// TIA Portal V20 export
// export: Created 2025-12-01T14:57:45.1353777Z, ExportSetting None, DisplayName Totally Integrated Automation Portal, DisplayVersion V20 Update 3, DisplayName TIA Portal Openness, DisplayVersion V20 Update 3, DisplayName TIA Portal Version Control Interface, DisplayVersion V20 Update 3, DisplayName STEP 7 Professional, DisplayVersion V20 Update 3, DisplayName STEP 7 Safety, DisplayVersion V20 Update 2, DisplayName WinCC Basic/Comfort/Advanced, DisplayVersion V20 Update 3, DisplayName WinCC Professional, DisplayVersion V20 Update 3, DisplayName WinCC Unified, DisplayVersion V20 Update 3
FUNCTION "FC783_Evento_BOET" : Void   // FC783, LAD
{ S7_Optimized_Access := 'FALSE' }
// stored: AutoNumber false, SetENOAutomatically false
   VAR_INPUT
      mensaje : Int;   // indice del array que estamos extrayendo
   END_VAR
   VAR_TEMP
      cero : Byte;
      retval : Int;
      pos_SSCC : UInt;
      Etiqueta_a_eliminar : ULInt;
      posicion_a_eliminar : UInt;
      cola : UInt;
      dato_actual_cola : UInt;
      pos_DB : UInt;
      registro_anterior : UInt;
      registro_siguiente : UInt;
      registro_etiqueta_limpio : "ROUT_Reg_Etiqueta";
   END_VAR
BEGIN

REGION Network 1 (SCL): INICIALIZACIONES
   REGION inicializacion

       // inicializamos las variables
       // 

       #retval := FILL(BVAL := #cero, BLK => #registro_etiqueta_limpio); // el registro de la etiqueta temporal



   END_REGION
END_REGION

REGION Network 2 (SCL): RECOJO Y CONVIERTO EL VALOR DE LA EITQUETA
   // buscamos donde empieza el SSCC en el mensaje y lo convertimos
   // 
   #pos_SSCC := FIND(IN1 := "DB199_eventos_convertidos".evento[#mensaje], IN2 := '[SSCC]');

   STRG_VAL(IN := "DB199_eventos_convertidos".evento[#mensaje],
            FORMAT := 0,
            P := (#pos_SSCC + 6), // +6 por lo que ocupa el atributo ['SSCC]'
            OUT => #Etiqueta_a_eliminar
   );

   // buscamos la etiqueta en la BBDD

   "FC715_Router_BuscarEtiqueta_Lint"(Etiqueta :=#Etiqueta_a_eliminar ,
                                      Posicion_BBDD => #posicion_a_eliminar);


   // si la posición a eliminar es 0, es que no existe ya en la BBDD y salimos de la función
   // 
   IF #posicion_a_eliminar = 0 THEN
       RETURN;
   END_IF;

     // si la hemos encontrado, además de eliminar la etiqueta, tenemos que mantener la coherencia
     // en el sistema de colas
     // para eso tenemos que mirar la posicón anterior y siguiente
     // 
     //
     //CALCULAMOS LA COLA A LA QUE PERTENECE LA ETIQUETA 
   #cola :=#Etiqueta_a_eliminar MOD "ROUT_N_Colas";


   REGION elegir_db_busqueda
       CASE #posicion_a_eliminar OF
           1..1000:
               #pos_DB := #posicion_a_eliminar;
               #registro_anterior:="DB201_RegEtiquetas_0001_1000".Reg_Etiqueta[#pos_DB].Anterior;
               #registro_siguiente:="DB201_RegEtiquetas_0001_1000".Reg_Etiqueta[#pos_DB].Posterior;
               // ahora que ya he sacado los datos necesarios limpio el registro
               "DB201_RegEtiquetas_0001_1000".Reg_Etiqueta[#pos_DB] := #registro_etiqueta_limpio;
               IF ((#registro_anterior = 0) AND (#registro_siguiente = 0)) THEN
                   "DB212_Cola_Activa".Cola[#cola] := 0;
                   RETURN;
               END_IF;

           1001..2000:
               #pos_DB := #posicion_a_eliminar - 1000;
               #registro_anterior := "DB202_RegEtiquetas_1001_2000".Reg_Etiqueta[#pos_DB].Anterior;
               #registro_siguiente := "DB202_RegEtiquetas_1001_2000".Reg_Etiqueta[#pos_DB].Posterior;
               "DB202_RegEtiquetas_1001_2000".Reg_Etiqueta[#pos_DB] := #registro_etiqueta_limpio;
               IF ((#registro_anterior = 0) AND (#registro_siguiente = 0)) THEN
                   "DB212_Cola_Activa".Cola[#cola] := 0;
                   RETURN;
               END_IF;

           2001..3000:
               #pos_DB := #posicion_a_eliminar - 2000;
              #registro_anterior:= "DB203_RegEtiquetas_2001_3000".Reg_Etiqueta[#pos_DB].Anterior ;
              #registro_siguiente:= "DB203_RegEtiquetas_2001_3000".Reg_Etiqueta[#pos_DB].Anterior;
               "DB203_RegEtiquetas_2001_3000".Reg_Etiqueta[#pos_DB] := #registro_etiqueta_limpio;
               // si los dos campos son 0 es que soy la unica etiqueta de la cola
               IF ((#registro_anterior = 0) AND (#registro_siguiente = 0)) THEN
                   "DB212_Cola_Activa".Cola[#cola] := 0;
                   RETURN;
               END_IF;
           3001..4000:
               #pos_DB := #posicion_a_eliminar - 3000;
               #registro_anterior := "DB204_RegEtiquetas_3001_4000".Reg_Etiqueta[#pos_DB].Anterior;
               #registro_siguiente := "DB204_RegEtiquetas_3001_4000".Reg_Etiqueta[#pos_DB].Posterior;
               "DB204_RegEtiquetas_3001_4000".Reg_Etiqueta[#pos_DB] := #registro_etiqueta_limpio;
               // si los dos campos son 0 es que soy la unica etiqueta de la cola
               IF ((#registro_anterior = 0) AND (#registro_siguiente = 0)) THEN
                   "DB212_Cola_Activa".Cola[#cola] := 0;
                   RETURN;
               END_IF;

               RETURN;
       END_CASE;
   END_REGION

   // si alguno de los dos datos es distinto de cero, tengo que recomponer la cola modificando
   // los registos de las etiquetas anteriores, posteriores y si procede la cola.
   // 

   IF #registro_anterior = 0 THEN
       // soy la primera de la cola y tengo que hacer que la que va despues de mi sea la primera de la cola

       "DB212_Cola_Activa".Cola[#cola] := #registro_siguiente;
   END_IF;

   //recomponemos registro anterior en la siguiente etiqueta
       REGION elegir_db_busqueda
           CASE #registro_siguiente OF
               0:
                   ;
               1..1000:
                   #pos_DB := #registro_siguiente;
                   "DB201_RegEtiquetas_0001_1000".Reg_Etiqueta[#pos_DB].Anterior := #registro_anterior;


               1001..2000:
                   #pos_DB := #registro_siguiente - 1000;
                   "DB202_RegEtiquetas_1001_2000".Reg_Etiqueta[#pos_DB].Anterior := #registro_anterior;

               2001..3000:
                   #pos_DB := #registro_siguiente - 2000;
                   "DB203_RegEtiquetas_2001_3000".Reg_Etiqueta[#pos_DB].Anterior := #registro_anterior;


               3001..4000:
                   #pos_DB := #registro_siguiente - 3000;
                   "DB204_RegEtiquetas_3001_4000".Reg_Etiqueta[#pos_DB].Anterior := #registro_anterior;


           END_CASE;
       END_REGION
       //recomponemos registro siguiente en la siguiente anterior
       REGION elegir_db_busqueda
           CASE #registro_anterior OF
               0:
                   ;
               1..1000:
                   #pos_DB := #registro_anterior;
                   "DB201_RegEtiquetas_0001_1000".Reg_Etiqueta[#pos_DB].Posterior := #registro_siguiente;
                   RETURN;

               1001..2000:
                   #pos_DB := #registro_anterior - 1000;
                   "DB202_RegEtiquetas_1001_2000".Reg_Etiqueta[#pos_DB].Posterior := #registro_siguiente;
                   RETURN;
               2001..3000:
                   #pos_DB := #registro_anterior - 2000;
                   "DB203_RegEtiquetas_2001_3000".Reg_Etiqueta[#pos_DB].Posterior := #registro_siguiente;
                   RETURN;

               3001..4000:
                   #pos_DB := #registro_anterior - 3000;
                   "DB204_RegEtiquetas_3001_4000".Reg_Etiqueta[#pos_DB].Posterior := #registro_siguiente;
                   RETURN;


           END_CASE;
       END_REGION
END_REGION
END_FUNCTION
